FUNCTION_BLOCK FB_CMS
VAR_INPUT
END_VAR
VAR_OUTPUT
	Impulse_X				:REAL;
	Impulse_Y				:REAL;
	Impulse_Z				:REAL;
	Temperature				:REAL;
END_VAR
VAR
	arrCMSData				AT %I*: ARRAY[0..19] OF BYTE;
	nChannelStatus			AT %I*: USINT;	
	
	AlarmTemperature		:BOOL;
	AlarmShock				:BOOL;
	AlarmRMS_PreMax			:BOOL;
	AlarmRMS_Max			:BOOL;
	
	ConfByte				:ARRAY[0..1] OF BYTE;
END_VAR


Impulse_X := FUN_ConvFourByteToReal32(nValue1 := arrCMSData[15], nValue2 := arrCMSData[14], nValue3 := arrCMSData[13], nValue4 := arrCMSData[12]); 
Impulse_Y := FUN_ConvFourByteToReal32(nValue1 := arrCMSData[11], nValue2 := arrCMSData[10], nValue3 := arrCMSData[9], nValue4 := arrCMSData[8]); 
Impulse_Z := FUN_ConvFourByteToReal32(nValue1 := arrCMSData[7], nValue2 := arrCMSData[6], nValue3 := arrCMSData[5], nValue4 := arrCMSData[4]); 
Temperature := FUN_ConvFourByteToReal32(nValue1 := arrCMSData[3], nValue2 := arrCMSData[2], nValue3 := arrCMSData[1], nValue4 := arrCMSData[0]); 



// Byte 18 - 19 is configureable byte. These can be set in SOPAS software.
ConfByte[0].0 := arrCMSData[18].0; // Deactivated
ConfByte[0].1 := arrCMSData[18].1; // Deactivated
ConfByte[0].2 := arrCMSData[18].2; // Deactivated
ConfByte[0].3 := arrCMSData[18].3; // Deactivated
ConfByte[0].4 := arrCMSData[18].4; // Deactivated
ConfByte[0].5 := arrCMSData[18].5; // Deactivated
ConfByte[0].6 := arrCMSData[18].6; // Deactivated
ConfByte[0].7 := arrCMSData[18].7; // Deactivated

ConfByte[1].0 := arrCMSData[19].0; // Deactivated
ConfByte[1].1 := arrCMSData[19].1; // Deactivated
ConfByte[1].2 := arrCMSData[19].2; // Deactivated
ConfByte[1].3 := arrCMSData[19].3; // Deactivated

AlarmTemperature := arrCMSData[19].4; 
AlarmShock := arrCMSData[19].5; 
AlarmRMS_PreMax := arrCMSData[19].6; 
AlarmRMS_Max := arrCMSData[19].7;

END_FUNCTION_BLOCK

(* stored: Version 1.1.0.1, ProductVersion 3.1.4024.12
   POU FB_CMS: Id {ce930956-c27d-48d7-8251-fdaf414d816b}, SpecialFunc None *)
